// Mitsubishi GX Works2 project: 실린더 제어하기4-2   PLC: Q03UDV

PROGRAM 01_MAIN
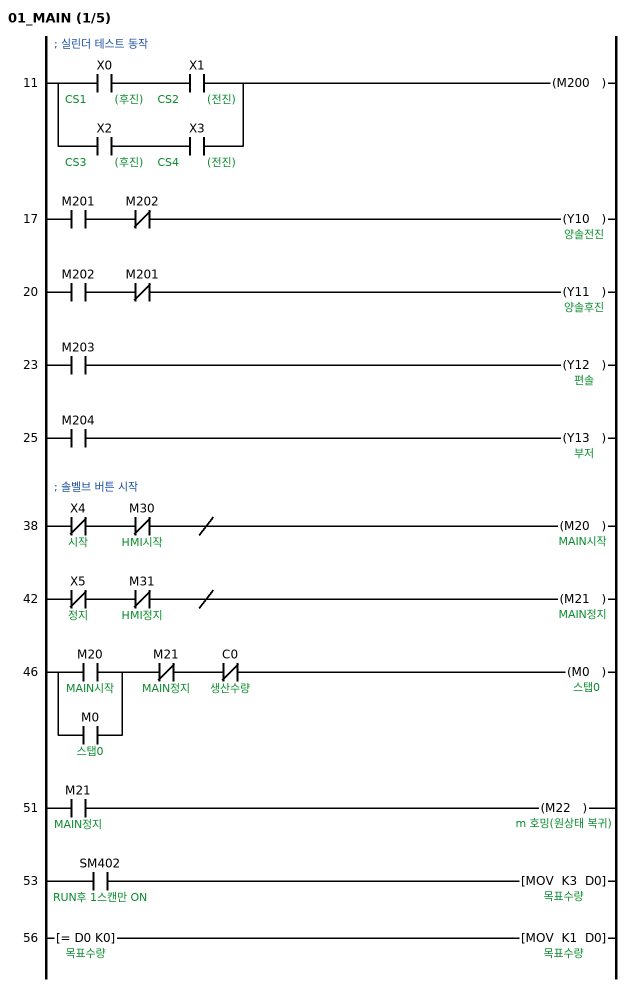
; 실린더 테스트 동작
11    LD      X0  ; CS1        (후진)
      AND     X1  ; CS2        (전진)
      LD      X2  ; CS3        (후진)
      AND     X3  ; CS4        (전진)
      ORB
      OUT     M200
17    LD      M201
      ANI     M202
      OUT     Y10  ; 양솔전진
20    LD      M202
      ANI     M201
      OUT     Y11  ; 양솔후진
23    LD      M203
      OUT     Y12  ; 편솔
25    LD      M204
      OUT     Y13  ; 부저
; 솔벨브 버튼 시작
38    LDI     X4  ; 시작
      ANI     M30  ; HMI시작
      INV
      OUT     M20  ; MAIN시작
42    LDI     X5  ; 정지
      ANI     M31  ; HMI정지
      INV
      OUT     M21  ; MAIN정지
46    LD      M20  ; MAIN시작
      OR      M0  ; 스탭0
      ANI     M21  ; MAIN정지
      ANI     C0  ; 생산수량
      OUT     M0  ; 스탭0
51    LD      M21  ; MAIN정지
      OUT     M22  ; m 호밍(원상태 복귀)
53    LD      SM402  ; RUN후 1스캔만 ON
      MOV     K3 D0  ; 목표수량
56    LD=     D0 K0  ; 목표수량
      MOV     K1 D0
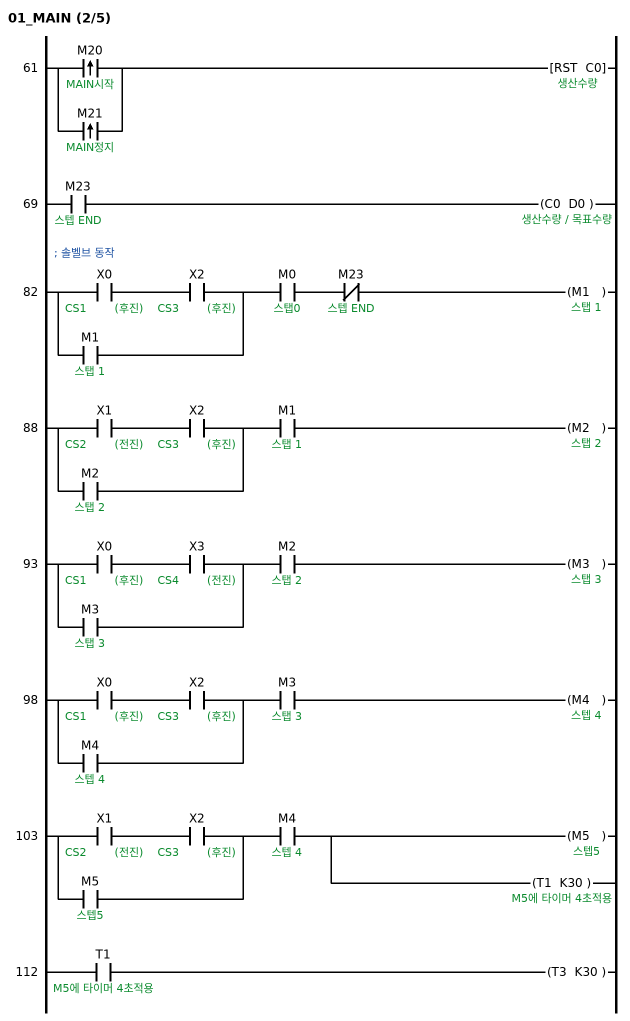
61    LDP     M20  ; MAIN시작
      ORP     M21  ; MAIN정지
      RST     C0  ; 생산수량
69    LD      M23  ; 스텝 END
      OUT     C0 D0  ; 생산수량 / 목표수량
; 솔벨브 동작
82    LD      X0  ; CS1        (후진)
      AND     X2  ; CS3        (후진)
      OR      M1  ; 스탭 1
      AND     M0  ; 스탭0
      ANI     M23  ; 스텝 END
      OUT     M1  ; 스탭 1
88    LD      X1  ; CS2        (전진)
      AND     X2  ; CS3        (후진)
      OR      M2  ; 스탭 2
      AND     M1  ; 스탭 1
      OUT     M2  ; 스탭 2
93    LD      X0  ; CS1        (후진)
      AND     X3  ; CS4        (전진)
      OR      M3  ; 스탭 3
      AND     M2  ; 스탭 2
      OUT     M3  ; 스탭 3
98    LD      X0  ; CS1        (후진)
      AND     X2  ; CS3        (후진)
      OR      M4  ; 스텝 4
      AND     M3  ; 스탭 3
      OUT     M4  ; 스텝 4
103   LD      X1  ; CS2        (전진)
      AND     X2  ; CS3        (후진)
      OR      M5  ; 스텝5
      AND     M4  ; 스텝 4
      OUT     M5  ; 스텝5
      OUT     T1 K30  ; M5에 타이머 4초적용
112   LD      T1  ; M5에 타이머 4초적용
      OUT     T3 K30
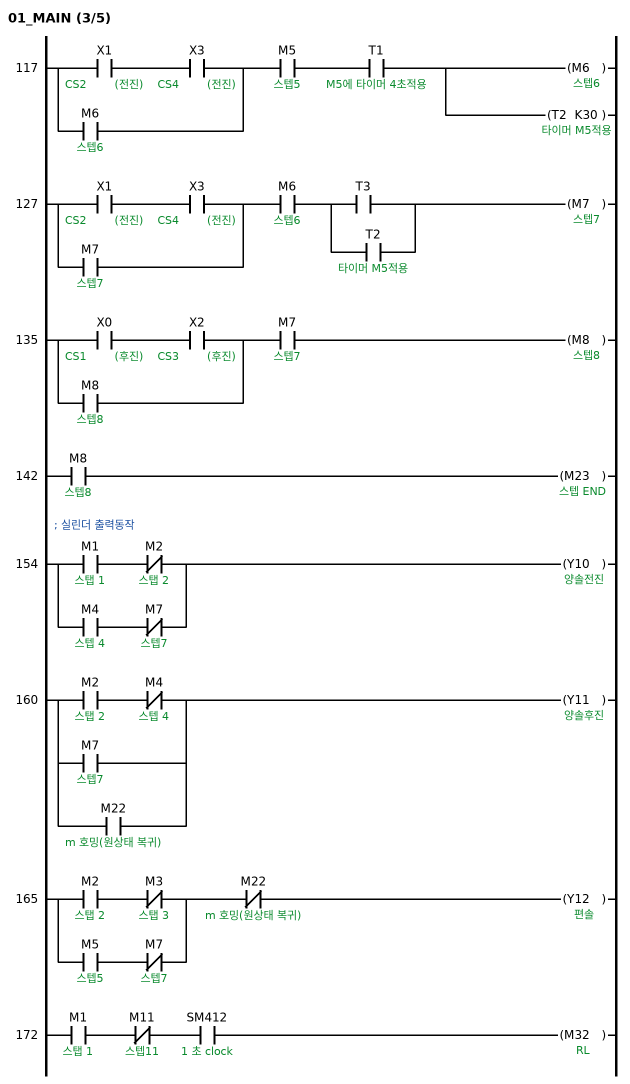
117   LD      X1  ; CS2        (전진)
      AND     X3  ; CS4        (전진)
      OR      M6  ; 스텝6
      AND     M5  ; 스텝5
      AND     T1  ; M5에 타이머 4초적용
      OUT     M6  ; 스텝6
      OUT     T2 K30  ; 타이머 M5적용
127   LD      X1  ; CS2        (전진)
      AND     X3  ; CS4        (전진)
      OR      M7  ; 스텝7
      AND     M6  ; 스텝6
      LD      T3
      OR      T2  ; 타이머 M5적용
      ANB
      OUT     M7  ; 스텝7
135   LD      X0  ; CS1        (후진)
      AND     X2  ; CS3        (후진)
      OR      M8  ; 스텝8
      AND     M7  ; 스텝7
      OUT     M8  ; 스텝8
; 
142   LD      M8  ; 스텝8
      OUT     M23  ; 스텝 END
; 실린더 출력동작
154   LD      M1  ; 스탭 1
      ANI     M2  ; 스탭 2
      LD      M4  ; 스텝 4
      ANI     M7  ; 스텝7
      ORB
      OUT     Y10  ; 양솔전진
160   LD      M2  ; 스탭 2
      ANI     M4  ; 스텝 4
      OR      M7  ; 스텝7
      OR      M22  ; m 호밍(원상태 복귀)
      OUT     Y11  ; 양솔후진
165   LD      M2  ; 스탭 2
      ANI     M3  ; 스탭 3
      LD      M5  ; 스텝5
      ANI     M7  ; 스텝7
      ORB
      ANI     M22  ; m 호밍(원상태 복귀)
      OUT     Y12  ; 편솔
172   LD      M1  ; 스탭 1
      ANI     M11  ; 스텝11
      AND     SM412  ; 1 초 clock
      OUT     M32  ; RL
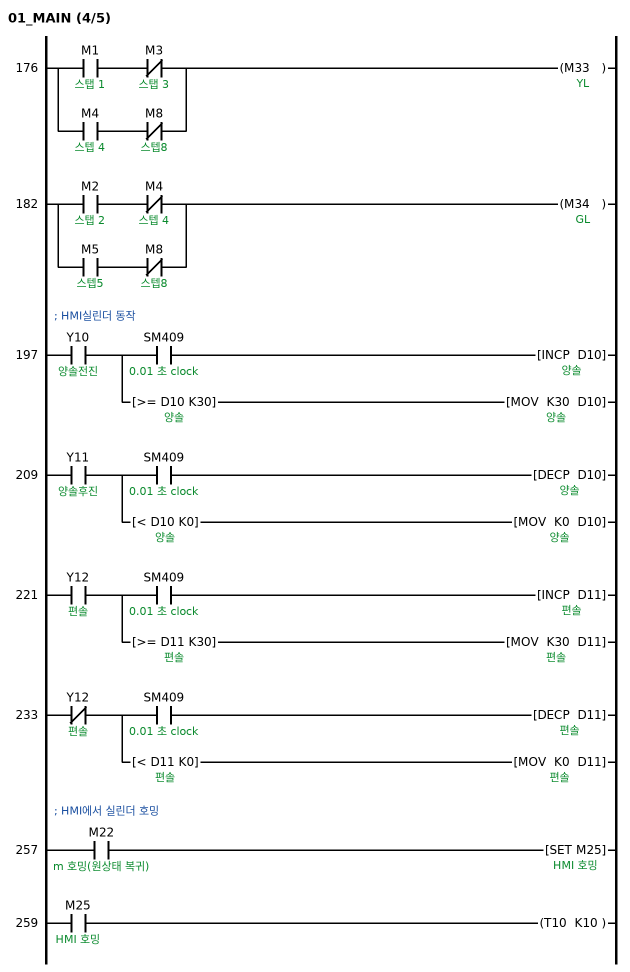
176   LD      M1  ; 스탭 1
      ANI     M3  ; 스탭 3
      LD      M4  ; 스텝 4
      ANI     M8  ; 스텝8
      ORB
      OUT     M33  ; YL
182   LD      M2  ; 스탭 2
      ANI     M4  ; 스텝 4
      LD      M5  ; 스텝5
      ANI     M8  ; 스텝8
      ORB
      OUT     M34  ; GL
; HMI실린더 동작
197   LD      Y10  ; 양솔전진
      MPS
      AND     SM409  ; 0.01 초 clock
      INCP    D10  ; 양솔
      MPP
      AND>=   D10 K30  ; 양솔
      MOV     K30 D10
209   LD      Y11  ; 양솔후진
      MPS
      AND     SM409  ; 0.01 초 clock
      DECP    D10
      MPP
      AND<    D10 K0  ; 양솔
      MOV     K0 D10
221   LD      Y12  ; 편솔
      MPS
      AND     SM409  ; 0.01 초 clock
      INCP    D11  ; 편솔
      MPP
      AND>=   D11 K30  ; 편솔
      MOV     K30 D11
233   LDI     Y12  ; 편솔
      MPS
      AND     SM409  ; 0.01 초 clock
      DECP    D11
      MPP
      AND<    D11 K0  ; 편솔
      MOV     K0 D11
; HMI에서 실린더 호밍
257   LD      M22  ; m 호밍(원상태 복귀)
      SET     M25  ; HMI 호밍
259   LD      M25  ; HMI 호밍
      OUT     T10 K10
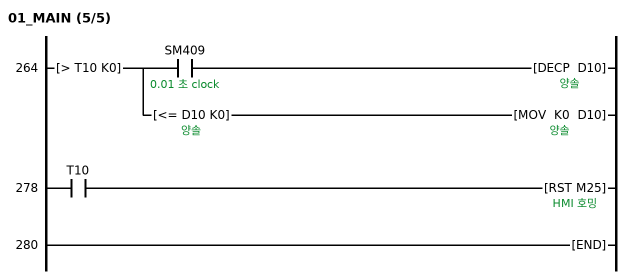
264   LD>     T10 K0
      MPS
      AND     SM409  ; 0.01 초 clock
      DECP    D10
      MPP
      AND<=   D10 K0  ; 양솔
      MOV     K0 D10
278   LD      T10
      RST     M25  ; HMI 호밍
280   END
END_PROGRAM

// device comments not shown above
M9  ; 스텝9
M10  ; 스텝10
M24  ; M_부저
D12  ; 스텝 번호
T0  ; 타이머
